FUNCTION_BLOCK Robot
VAR_INPUT
	enable: BOOL;
	vXref, vYref, vThetaRef: LREAL;
END_VAR
VAR_OUTPUT
	vX, vY, vTheta: LREAL;
END_VAR
VAR
	//inputs to robot
	vXtoRobot 		AT%Q*: LREAL;
	vYtoRobot		AT%Q*: LREAL;
	vThetaToRobot 	AT%Q*: LREAL;
	
	//outputs from robot
	vXfromRobot 		AT%I*: LREAL;
	vYfromRobot			AT%I*: LREAL;
	vThetaFromRobot 	AT%I*: LREAL;
END_VAR

//write control outputs to robot if enabled
IF enable = TRUE THEN
			vXtoRobot     := vXref;
			vYtoRobot	  := vYref;
			vThetaToRobot := vThetaRef;
ELSE
			vXtoRobot     := 0;
			vYtoRobot	  := 0;
			vThetaToRobot := 0;
END_IF

END_FUNCTION_BLOCK

(* stored: Version 1.1.0.1, ProductVersion 3.1.4024.11
   POU Robot: Id {c2c95814-6e9d-4a67-9cd4-cf68c7267fb5}, SpecialFunc None *)
